FUNCTION_BLOCK FB_Blink
VAR_INPUT
	bEnable : BOOL := FALSE;         // Enables the blink
    tPeriod : TIME := T#1S;       	// cycle total time (on + off)
END_VAR
VAR_OUTPUT
	bBlink : BOOL;                   // blinking output
END_VAR
VAR
	ton : TON;
END_VAR

// State alternation every tPeriod/2
IF bEnable THEN
    ton(IN := NOT ton.Q, PT := tPeriod / 2);
    ton(IN := TRUE);
    
    IF ton.Q THEN
        bBlink := NOT bBlink;
        ton(IN := FALSE);  // resets the cycle
    END_IF;
ELSE
    ton(IN := FALSE);
    bBlink := FALSE;
END_IF;

END_FUNCTION_BLOCK

(* stored: Version 1.1.0.1, ProductVersion 3.1.4024.12
   POU FB_Blink: Id {2252363c-dbe1-4a37-984a-e77f414499c2}, SpecialFunc None *)
